INTERFACE I_AssetState EXTENDS I_Observer

METHOD execute_on_state : BOOL
VAR_INPUT
END_VAR
END_METHOD

END_INTERFACE

(* stored: Version 1.1.0.1, ProductVersion 3.1.4026.13
   Itf I_AssetState: Id {ec05e055-f1f5-494a-9dff-ceb0dd092a60}
   Method execute_on_state: Id {2abae85d-9c48-4462-a344-622519f466d9} *)
